(* PLC project Unnamed, Unknown Unnamed 1 *)
(* stored: creationDateTime 2021-05-11T15:41:27, modificationDateTime 2021-08-18T14:56:07 *)

PROGRAM RCP_PLC
  VAR
    TIME_IN AT %MD0 : REAL;
    TIME_OUT AT %MD1 : REAL;
    RCP_FLOW AT %MD2 : REAL;
    RCP_PUMP_SPEED AT %MD3 : REAL;
    MANIPIO_CONTROL AT %MD4 : REAL := 0.0;
    KPI AT %MD5 : REAL := 0.001;
    Ti AT %MD6 : REAL := 30.0;
    SET_POINT AT %MD7 : REAL := 8801.4;
    INIT AT %MD8 : REAL := 90.0;
  END_VAR
  VAR
    INTEGRAL0 : INTEGRAL;
  END_VAR
  VAR  (* added by the conversion: wires and edge detectors of the diagram *)
    _MUL7_OUT : REAL;
    _LIMIT18_OUT : ANY;
    _ADD14_OUT : ANY;
  END_VAR

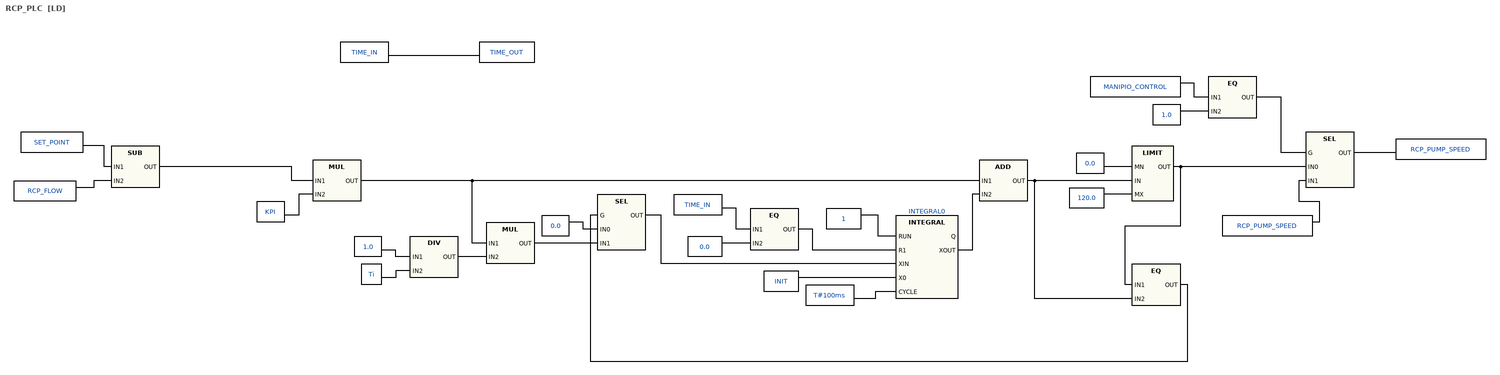
(* LD diagram, written out as Structured Text *)
TIME_OUT := TIME_IN;
_MUL7_OUT := (SET_POINT - RCP_FLOW) * KPI;
INTEGRAL0(RUN := 1, R1 := TIME_IN = 0.0, XIN := SEL(_LIMIT18_OUT = _ADD14_OUT, 0.0, _MUL7_OUT * (1.0 / Ti)), X0 := INIT, CYCLE := T#100ms);
_ADD14_OUT := _MUL7_OUT + INTEGRAL0.XOUT;
_LIMIT18_OUT := LIMIT(0.0, _ADD14_OUT, 120.0);
RCP_PUMP_SPEED := SEL(MANIPIO_CONTROL = 1.0, _LIMIT18_OUT, RCP_PUMP_SPEED);
END_PROGRAM

CONFIGURATION Config0
  RESOURCE Res0 ON PLC
    TASK task0(INTERVAL := T#100ms, PRIORITY := 0);
    PROGRAM instance0 WITH task0 : RCP_PLC;
  END_RESOURCE
END_CONFIGURATION
